TYPE DUT_MotionPneumaticActuator : ST_MotionPneumaticActuator; END_TYPE

(* stored: Version 1.1.0.1
   DUT DUT_MotionPneumaticActuator: Id {9d6f4ada-511a-43b4-beed-b74155f0ce83} *)
